INTERFACE itfSynchronizedAxisCommand EXTENDS itfAxisCommand

PROPERTY InSync : BOOL
GET
END_GET
END_PROPERTY

END_INTERFACE

(* stored: Version 1.1.0.1, ProductVersion 3.1.4024.11
   Itf itfSynchronizedAxisCommand: Id {0afa7a1b-cb9a-4e83-a79a-3a7500d345c7}
   Property InSync: Id {1cebdef4-5269-4b19-9ab8-4bf47a5d803e}
   Get Get: Id {d74ec274-98ae-4900-ae6c-83710ca6dd85} *)
